PROGRAM MAIN
VAR
END_VAR

ProcessLamp();
FullProcess();
ShortProcess(); 
FeedMotor1Manualcontrol();
CabinetSwitch();
ValveManualControl();
Scaling();
FeedMotor2Manualcontrol();
RemovalProgram();

END_PROGRAM

(* stored: Version 1.1.0.1, ProductVersion 3.1.4024.12
   POU MAIN: Id {552b854d-2ec7-4dbd-af65-fc6da06c4304}, SpecialFunc None *)
